INTERFACE I_StationProcess

PROPERTY SetOpMode : E_OpMode
SET
END_SET
END_PROPERTY

PROPERTY State : E_StationProcessState
GET
END_GET
SET
END_SET
END_PROPERTY

METHOD Update
VAR_INPUT
	iStation : I_XTS_Station_PLC;	
END_VAR
END_METHOD

END_INTERFACE

(* stored: Version 1.1.0.1, ProductVersion 3.1.4024.12
   Itf I_StationProcess: Id {186b54bc-4cfe-4388-a319-b3213386405b}
   Property SetOpMode: Id {ce96595a-cc7b-45eb-9684-4d775a0b6136}
   Set Set: Id {104f3592-9932-4629-9328-28cb58cfd36e}
   Property State: Id {893fa886-f71f-49d4-b79f-41ce9b10ddb8}
   Get Get: Id {f9b4a8d9-39f5-4ac1-b692-cb7caa168642}
   Set Set: Id {6361f94d-3861-47a5-bfb0-4cd95f6738da}
   Method Update: Id {98b90e30-ef9e-42d9-ba1b-b560b7f75cb0} *)
